// TIA Portal V18 export
FUNCTION_BLOCK "auto_analog_NORMAL"   // FB5, FBD
{ S7_Optimized_Access := 'TRUE' }
VERSION : 0.1
// stored: AutoNumber true, IsIECCheckEnabled false, IsRetainMemResEnabled false, MemoryReserve 100, SetENOAutomatically false, UDAEnableTagReadback false
   VAR_INPUT
      ALLOWED : Bool;
      MultiTurnGoesFwdOnly : Bool;
      isMultiturn : Bool;
      arrived_missed : Bool;
      SET_SPD_ABS : Real;
      POS : Real;
      TARGET : Real;
      FOLLOW : Bool;
      xFwdOK : Bool;
      xRevOK : Bool;
      par_spd_absmax : Real;
      par_dist_absMax : Real;
      par_spd_crawl : Real;
      par_dist_crawl : Real;
      par_dist_stop : Real;
      par_lim_fwd : Real;
      par_lim_rev : Real;
      par_prec_au : Real;
      par_tout_follw : Time;
      par_t_acc : Real;
   END_VAR
   VAR_OUTPUT
      SPEED : Real;
      INPOS : Bool;
      ER_follow : Bool;
      ER_settings : Bool;
      ER : Bool;
      erws : WString;
   END_VAR
   VAR
      SET_SPD_ABS_slowlyaccelerated { ExternalAccessible := 'False'; ExternalVisible := 'False'; ExternalWritable := 'False'} : Real;
      should_go { ExternalAccessible := 'False'; ExternalVisible := 'False'; ExternalWritable := 'False'} : Bool;
      mot_speed_slowly_accelerated_Instance { S7_SetPoint := 'True'} : "mot_speed_abs_slowly_accelerated";
      mot_speed_wdir_slowly_accelerated_Instance { S7_SetPoint := 'True'} : "mot_speed_wdir_slowly_accelerated";
      arrived1 { S7_SetPoint := 'True'} : "mot_auto_calc_arrivedFB";
      arrived2 { S7_SetPoint := 'True'} : "mot_auto_calc_arrivedFB";
      arrived3 { S7_SetPoint := 'True'} : "mot_auto_calc_arrivedFB";
      IEC_Timer_0_Instance { S7_SetPoint := 'True'} : TOF_TIME;
   END_VAR
   VAR_TEMP
      dir_fwd : Bool;
      dir_rev : Bool;
      arrived : Bool;
      speed_calculated : Real;
      speed_limited_fwd : Real;
      speed_limited_rev : Real;
      distance : Real;
      speed_limited_by_target_slowlychanging : Real;
      speed_limited_by_target : Real;
      estop_ok_no_err : Bool;
      speed_calc_abs : Real;
      speed_w_direction : Real;
      stop_now : Bool;
      ER_w : WString;
      length : Real;
      delta : Real;
      delta_minus : Real;
   END_VAR
   VAR CONSTANT
      erws_noer : WString := WSTRING#'';
      erws_1 : WString := WSTRING#'stuck fwd';
      erws_2 : WString := WSTRING#'stuck rev';
      erws_5 : WString := WSTRING#'->+';
      erws_4 : WString := WSTRING#'fast<0';
      erws_3 : WString := WSTRING#'fst<slo';
      erws_6 : WString := WSTRING#'tOUT<=0';
   END_VAR
   VAR_TEMP   // added for the SCL form of the ladder/FBD networks
      _w1 : Bool;
      _w2 : Bool;
      _w3 : Bool;
      _w4 : Bool;
   END_VAR
BEGIN

REGION Network 1
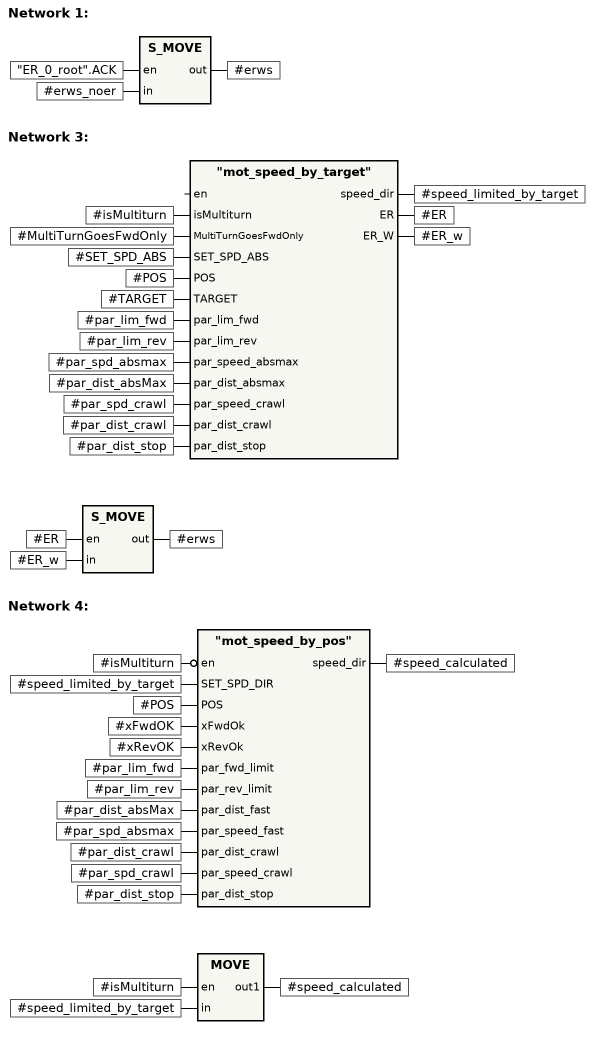
   IF "ER_0_root".ACK THEN #erws := #erws_noer; END_IF;
END_REGION

REGION Network 3
   "mot_speed_by_target"(isMultiturn := #isMultiturn,
                         MultiTurnGoesFwdOnly := #MultiTurnGoesFwdOnly,
                         SET_SPD_ABS := #SET_SPD_ABS,
                         POS := #POS,
                         TARGET := #TARGET,
                         par_lim_fwd := #par_lim_fwd,
                         par_lim_rev := #par_lim_rev,
                         par_speed_absmax := #par_spd_absmax,
                         par_dist_absmax := #par_dist_absMax,
                         par_speed_crawl := #par_spd_crawl,
                         par_dist_crawl := #par_dist_crawl,
                         par_dist_stop := #par_dist_stop,
                         speed_dir => #speed_limited_by_target,
                         ER => #ER,
                         ER_W => #ER_w);
   IF #ER THEN #erws := #ER_w; END_IF;
END_REGION

REGION Network 4
   IF NOT #isMultiturn THEN
       "mot_speed_by_pos"(SET_SPD_DIR := #speed_limited_by_target,
                          POS := #POS,
                          xFwdOk := #xFwdOK,
                          xRevOk := #xRevOK,
                          par_fwd_limit := #par_lim_fwd,
                          par_rev_limit := #par_lim_rev,
                          par_dist_fast := #par_dist_absMax,
                          par_speed_fast := #par_spd_absmax,
                          par_dist_crawl := #par_dist_crawl,
                          par_speed_crawl := #par_spd_crawl,
                          par_dist_stop := #par_dist_stop,
                          speed_dir => #speed_calculated);
   END_IF;
   IF #isMultiturn THEN #speed_calculated := #speed_limited_by_target; END_IF;
END_REGION

REGION Network 5
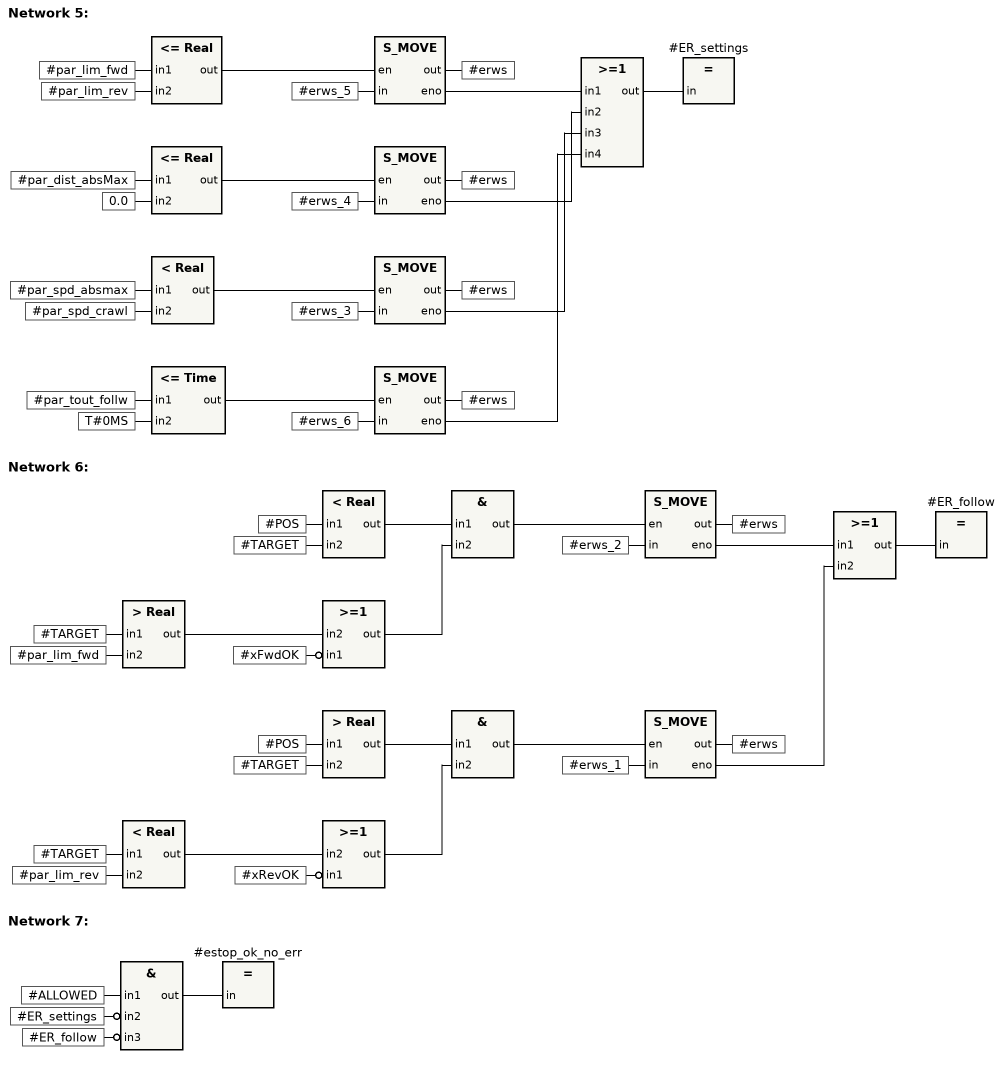
   #_w1 := #par_lim_fwd <= #par_lim_rev;
   IF #_w1 THEN #erws := #erws_5; END_IF;
   #_w2 := #par_dist_absMax <= 0.0;
   IF #_w2 THEN #erws := #erws_4; END_IF;
   #_w3 := #par_spd_absmax < #par_spd_crawl;
   IF #_w3 THEN #erws := #erws_3; END_IF;
   #_w4 := #par_tout_follw <= T#0MS;
   IF #_w4 THEN #erws := #erws_6; END_IF;
   #ER_settings := #_w1 OR #_w2 OR #_w3 OR #_w4;
END_REGION

REGION Network 6
   #_w1 := (#POS < #TARGET) AND ((#TARGET > #par_lim_fwd) OR NOT #xFwdOK);
   IF #_w1 THEN #erws := #erws_2; END_IF;
   #_w2 := (#POS > #TARGET) AND ((#TARGET < #par_lim_rev) OR NOT #xRevOK);
   IF #_w2 THEN #erws := #erws_1; END_IF;
   #ER_follow := #_w1 OR #_w2;
END_REGION

REGION Network 7
   #estop_ok_no_err := #ALLOWED AND NOT #ER_settings AND NOT #ER_follow;
END_REGION

REGION Network 8 (SCL)
   IF #isMultiturn THEN
       #length := ABS(#par_lim_fwd - #par_lim_rev);
       #delta := #length;
   ELSE
       #delta := 0    ;
   END_IF;
   #delta_minus := -#delta;
END_REGION

REGION Network 9
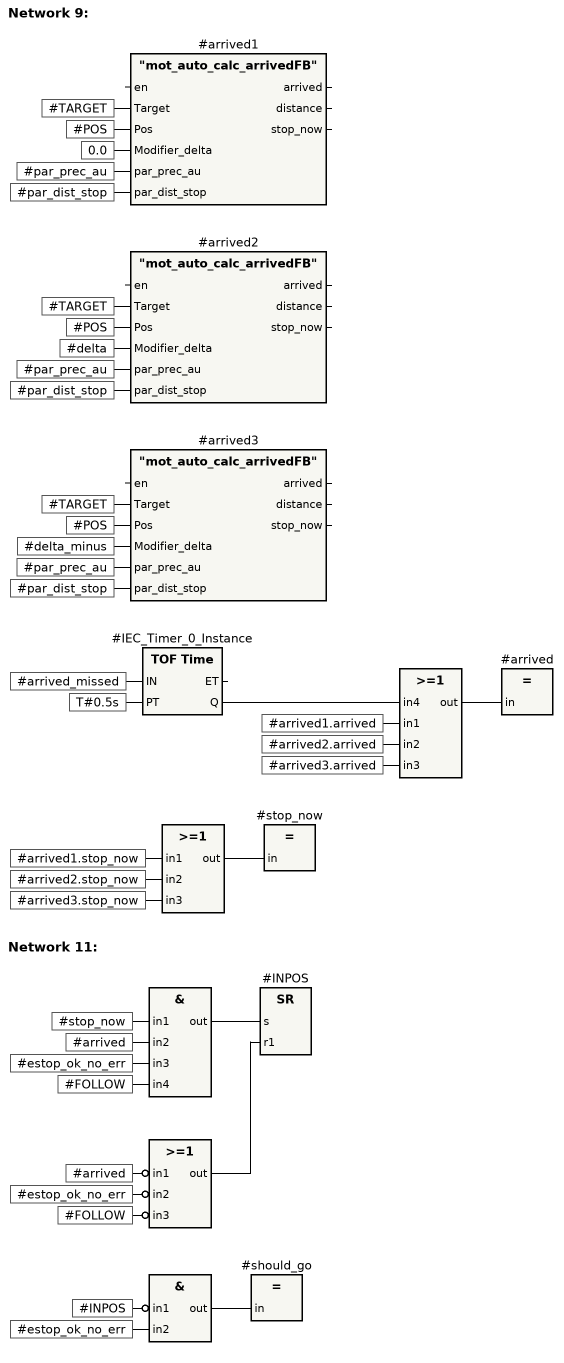
   #arrived1(Target := #TARGET,   // "mot_auto_calc_arrivedFB"
             Pos := #POS,
             Modifier_delta := 0.0,
             par_prec_au := #par_prec_au,
             par_dist_stop := #par_dist_stop);
   #arrived2(Target := #TARGET,   // "mot_auto_calc_arrivedFB"
             Pos := #POS,
             Modifier_delta := #delta,
             par_prec_au := #par_prec_au,
             par_dist_stop := #par_dist_stop);
   #arrived3(Target := #TARGET,   // "mot_auto_calc_arrivedFB"
             Pos := #POS,
             Modifier_delta := #delta_minus,
             par_prec_au := #par_prec_au,
             par_dist_stop := #par_dist_stop);
   #IEC_Timer_0_Instance(IN := #arrived_missed, PT := T#0.5s);   // TOF
   #arrived := #IEC_Timer_0_Instance.Q OR #arrived1.arrived OR #arrived2.arrived OR #arrived3.arrived;
   #stop_now := #arrived1.stop_now OR #arrived2.stop_now OR #arrived3.stop_now;
END_REGION

REGION Network 11
   IF #stop_now AND #arrived AND #estop_ok_no_err AND #FOLLOW THEN
       #INPOS := TRUE;   // SR flip-flop
   END_IF;
   IF NOT #arrived OR NOT #estop_ok_no_err OR NOT #FOLLOW THEN #INPOS := FALSE; END_IF;
   #should_go := NOT #INPOS AND #estop_ok_no_err;
END_REGION

REGION Network 12
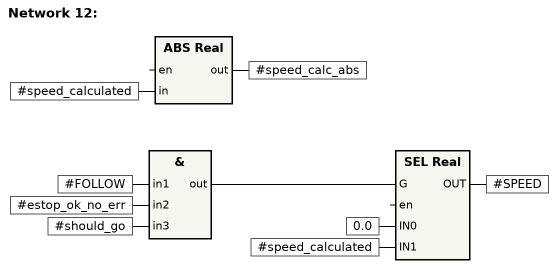
   #speed_calc_abs := ABS(#speed_calculated);
   #SPEED := SEL(G := #FOLLOW AND #estop_ok_no_err AND #should_go, IN0 := 0.0, IN1 := #speed_calculated);
END_REGION
END_FUNCTION_BLOCK
